Fanuc KAREL source: SET_TIME.kl

PROGRAM T
%NOLOCKGROUP
VAR
 v0 : INTEGER
BEGIN
 SET_TIME(v0)
END T
